Omron CX-Programmer project NuevoProyecto (CX-Programmer 9.61)

# PLC TunelDosTrenes: CJ2M CPU11

## Program NuevoPrograma1 (cyclic task 0)
Local symbols
Aproximación1 0.12 BOOL  ; 0.12
Aproximación2 0.14 BOOL  ; 0.14
Espera1 0.10 BOOL
Espera2 0.11 BOOL
P0 2.00 BOOL
P1 2.01 BOOL
P2 2.02 BOOL
P3 2.03 BOOL
P4 2.04 BOOL
P5 2.05 BOOL
P6 2.06 BOOL
Rojo1 1.08 BOOL  ; 1.08
Rojo2 1.09 BOOL  ; 1.09
Salida1 0.13 BOOL  ; 0.13
Salida2 0.15 BOOL  ; 0.15
Verde1 1.00 BOOL  ; 1.00
Verde2 1.01 BOOL  ; 1.01

### Section main

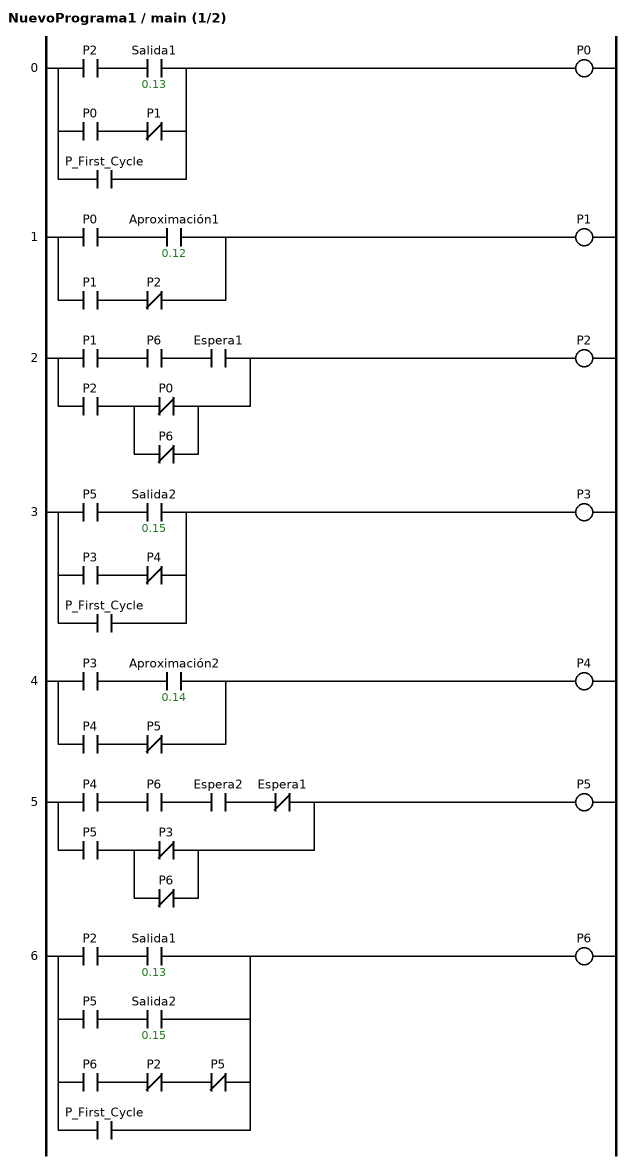
; rung 0
LD P2
AND Salida1  ; 0.13
LD P0
ANDNOT P1
ORLD
OR P_First_Cycle
OUT P0
; rung 1
LD P0
AND Aproximación1  ; 0.12
LD P1
ANDNOT P2
ORLD
OUT P1
; rung 2
LD P1
AND P6
AND Espera1
LD P2
LDNOT P0
ORNOT P6
ANDLD
ORLD
OUT P2
; rung 3
LD P5
AND Salida2  ; 0.15
LD P3
ANDNOT P4
ORLD
OR P_First_Cycle
OUT P3
; rung 4
LD P3
AND Aproximación2  ; 0.14
LD P4
ANDNOT P5
ORLD
OUT P4
; rung 5
LD P4
AND P6
AND Espera2
ANDNOT Espera1
LD P5
LDNOT P3
ORNOT P6
ANDLD
ORLD
OUT P5
; rung 6
LD P2
AND Salida1  ; 0.13
LD P5
AND Salida2  ; 0.15
ORLD
LD P6
ANDNOT P2
ANDNOT P5
ORLD
OR P_First_Cycle
OUT P6

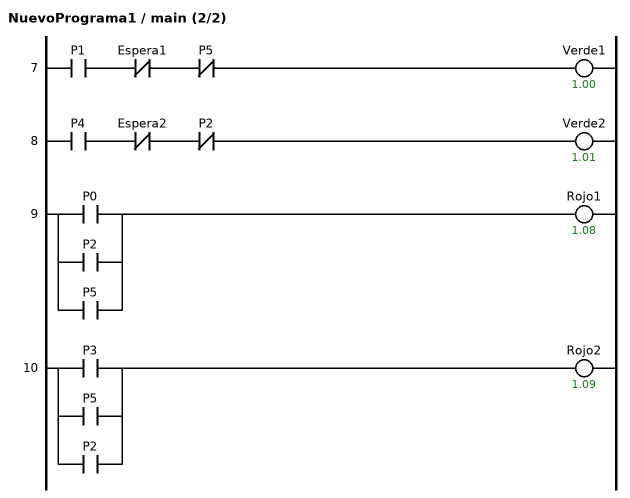
; rung 7
LD P1
ANDNOT Espera1
ANDNOT P5
OUT Verde1  ; 1.00
; rung 8
LD P4
ANDNOT Espera2
ANDNOT P2
OUT Verde2  ; 1.01
; rung 9
LD P0
OR P2
OR P5
OUT Rojo1  ; 1.08
; rung 10
LD P3
OR P5
OR P2
OUT Rojo2  ; 1.09

### Section END
; rung 0
END(001)